PROGRAM MAIN
VAR
	_ST80a		: ST80a;
	_ST80b		: sT80b; 
	_ST80c		: ST80c; 
END_VAR

_ST80a._Ready();

END_PROGRAM

(* stored: Version 1.1.0.1, ProductVersion 3.1.4024.12
   POU MAIN: Id {cda09ef7-7100-4d20-8a2f-028dec4c33fa}, SpecialFunc None *)
